// TIA Portal project "Modbus TCP with RFID_V15" (V15)

(* hardware
DEVICE "S7-1200 station_1"  S7-1200 Station
   slot 0: "Rack_0"  Rack  V1.0
   slot 1: "mbClient"  CPU 1215C DC/DC/DC  6ES7 215-1AG40-0XB0  V4.2
*)

// ===== PLC "mbClient"  CPU 1215C DC/DC/DC =====

VAR_GLOBAL   // PLC tag table "默认变量表"
   "System_Byte" AT %MB1 : Byte;
   "FirstScan" AT %M1.0 : Bool;
   "DiagStatusUpdate" AT %M1.1 : Bool;
   "AlwaysTRUE" AT %M1.2 : Bool;
   "AlwaysFALSE" AT %M1.3 : Bool;
   "ReqClient_1" AT %M0.0 : Bool;
   "DisConnect" AT %M0.1 : Bool;
   "DoneClient_1" AT %M0.2 : Bool;
   "BusyClient_1" AT %M0.3 : Bool;
   "ErrorClient_1" AT %M0.4 : Bool;
   "StatusClient_1" AT %MW2 : Word;
   "ReqClient_2" AT %M4.0 : Bool;
   "DoneClient_2" AT %M4.1 : Bool;
   "BusyClient_2" AT %M4.2 : Bool;
   "ErrorClient_2" AT %M4.3 : Bool;
   "StatusClient_2" AT %MW6 : Word;
   "Connected_P" AT %M8.0 : Bool;
   "ReqClientable_1" AT %M9.0 : Bool;
   "ReqClientable_2" AT %M9.1 : Bool;
   "ReqClientMid_1" AT %M9.2 : Bool;
   "ReqClientMid_2" AT %M9.3 : Bool;
   "ReqClientTimeIN_1" AT %MD50 : Time;
   "ReqClientTimeIN_1(1)" AT %MD54 : Time;
   "ReqClientTimeOUT_1" AT %MD58 : Time;
   "ReqClientTimeOUT_1(1)" AT %MD62 : Time;
   "ReqClientTimeIN_2" AT %MD66 : Time;
   "ReqClientTimeIN_2(1)" AT %MD70 : Time;
   "ReqClientTimeOUT_2" AT %MD74 : Time;
   "ReqClientTimeOUT_2(1)" AT %MD78 : Time;
END_VAR

DATA_BLOCK "MyModbusTcp"   // DB1
{ S7_Optimized_Access := 'TRUE' }
VERSION : 0.1
   VAR
      Connect : TCON_IP_v4;
   END_VAR
BEGIN
   Connect.InterfaceId := 64;
   Connect.ID := 16#01;
   Connect.ConnectionType := 16#0B;
   Connect.ActiveEstablished := TRUE;
   Connect.RemoteAddress.ADDR[1] := 192;
   Connect.RemoteAddress.ADDR[2] := 168;
   Connect.RemoteAddress.ADDR[3] := 0;
   Connect.RemoteAddress.ADDR[4] := 100;
   Connect.RemotePort := 502;
END_DATA_BLOCK

// folder: System blocks/Program resources

DATA_BLOCK "IEC_Timer_0_DB"   // DB3
{ S7_Optimized_Access := 'TRUE' }
AUTHOR : Simatic
FAMILY : IEC
NAME : IEC_TMR
VERSION : 1.0
// stored: InstanceOfName IEC_TIMER
"IEC_TIMER"
BEGIN
END_DATA_BLOCK

DATA_BLOCK "IEC_Timer_0_DB_1"   // DB4
{ S7_Optimized_Access := 'TRUE' }
AUTHOR : Simatic
FAMILY : IEC
NAME : IEC_TMR
VERSION : 1.0
// stored: InstanceOfName IEC_TIMER
"IEC_TIMER"
BEGIN
END_DATA_BLOCK

DATA_BLOCK "IEC_Timer_0_DB_2"   // DB5
{ S7_Optimized_Access := 'TRUE' }
AUTHOR : Simatic
FAMILY : IEC
NAME : IEC_TMR
VERSION : 1.0
// stored: InstanceOfName IEC_TIMER
"IEC_TIMER"
BEGIN
END_DATA_BLOCK

DATA_BLOCK "IEC_Timer_0_DB_3"   // DB6
{ S7_Optimized_Access := 'TRUE' }
AUTHOR : Simatic
FAMILY : IEC
NAME : IEC_TMR
VERSION : 1.0
// stored: InstanceOfName IEC_TIMER
"IEC_TIMER"
BEGIN
END_DATA_BLOCK

// folder: (top level)

ORGANIZATION_BLOCK "Main"   // OB1, LAD, ProgramCycle
TITLE = "Main Program Sweep (Cycle)"
{ S7_Optimized_Access := 'TRUE' }
VERSION : 0.1
// S7-1215C as client，S7-1215C Read RFID 40001~40007 data and Save to MW100 ~ MW114
   VAR_INPUT
      Initial_Call : Bool;   // Initial call of this OB
      Remanence : Bool;   // =True, if remanent data are available
   END_VAR
BEGIN

REGION Network 1: Check Modbus TCP Connect Status
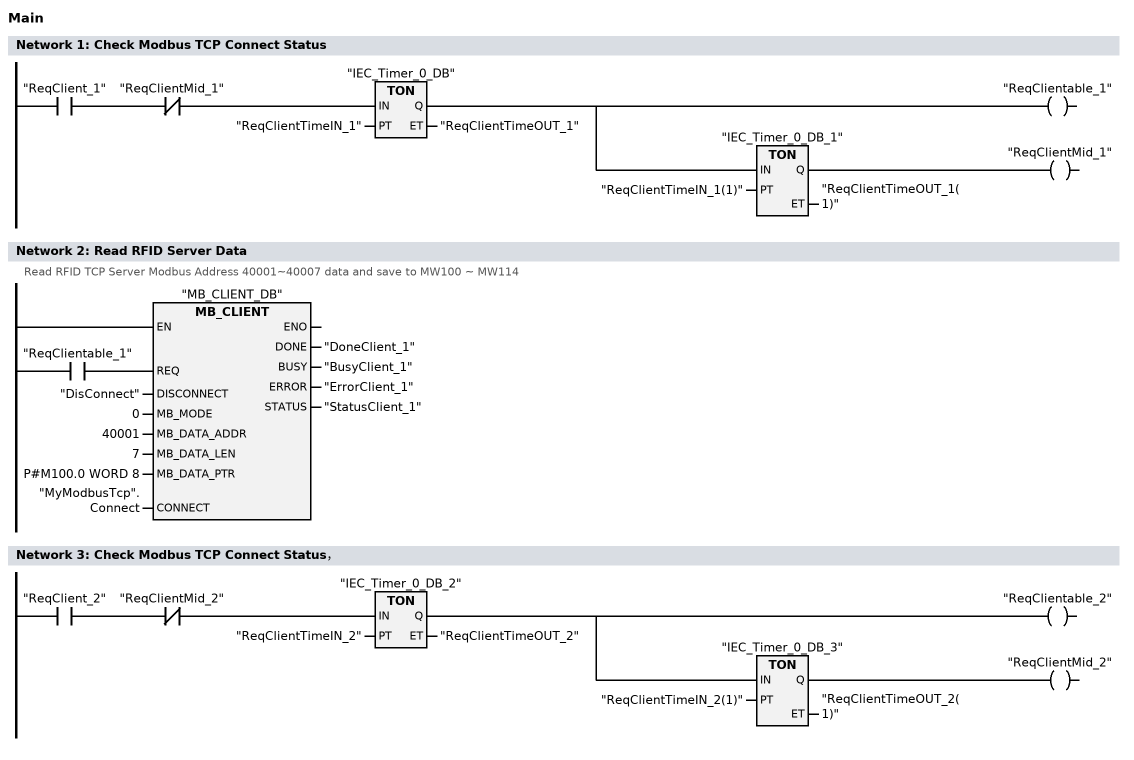
   "IEC_Timer_0_DB".TON(IN := "ReqClient_1" AND NOT "ReqClientMid_1",
                        PT := "ReqClientTimeIN_1",
                        ET => "ReqClientTimeOUT_1");
   "ReqClientable_1" := "IEC_Timer_0_DB".Q;
   "IEC_Timer_0_DB_1".TON(IN := "IEC_Timer_0_DB".Q, PT := "ReqClientTimeIN_1(1)", ET => "ReqClientTimeOUT_1(1)");
   "ReqClientMid_1" := "IEC_Timer_0_DB_1".Q;
END_REGION

REGION Network 2: Read RFID Server Data
   // Read RFID TCP Server Modbus Address 40001~40007 data and save to MW100 ~ MW114
   "MB_CLIENT_DB"(REQ := "ReqClientable_1",   // MB_CLIENT
                  DISCONNECT := "DisConnect",
                  MB_MODE := 0,
                  MB_DATA_ADDR := 40001,
                  MB_DATA_LEN := 7,
                  MB_DATA_PTR := P#M100.0 WORD 8,
                  CONNECT := "MyModbusTcp".Connect,
                  DONE => "DoneClient_1",
                  BUSY => "BusyClient_1",
                  ERROR => "ErrorClient_1",
                  STATUS => "StatusClient_1");
END_REGION

REGION Network 3: Check Modbus TCP Connect Status，
   "IEC_Timer_0_DB_2".TON(IN := "ReqClient_2" AND NOT "ReqClientMid_2",
                          PT := "ReqClientTimeIN_2",
                          ET => "ReqClientTimeOUT_2");
   "ReqClientable_2" := "IEC_Timer_0_DB_2".Q;
   "IEC_Timer_0_DB_3".TON(IN := "IEC_Timer_0_DB_2".Q,
                          PT := "ReqClientTimeIN_2(1)",
                          ET => "ReqClientTimeOUT_2(1)");
   "ReqClientMid_2" := "IEC_Timer_0_DB_3".Q;
END_REGION
END_ORGANIZATION_BLOCK